{attribute 'qualified_only'}
VAR_GLOBAL
END_VAR

(* stored: Version 1.1.0.1, ProductVersion 3.1.4024.10
   GVL HMI: Id {0ad82c49-6696-452a-b345-303f9f782f73} *)
